FUNCTION_BLOCK OPCUA_WRITE_1322467A4CC663E9C (* Generic Interface Function Block Type *)
  (* Standard: 61499-2 *)
  (* Version 0.0, 01/09/2020, Administrator, nxtControl GmbH, Template *)
  PACKAGE Main;
  (* Compiler Cpp nxtControl builtin 1.0 *)
  {SET_ATTRIBUTE(Runtime.FBType.ImplementingType, Standard.OPCUAClient#DYNGEN_OPCUA_WRITE)}
  {SET_ATTRIBUTE(Configuration.GenericFBType.InterfaceParams, Standard.OPCUAClient#CNTX:=2;VALUE${CNTX$}:BOOL,BOOL)}
  {SET_ATTRIBUTE(Configuration.FBType.IsKind.OPCUA_CLIENT, )}
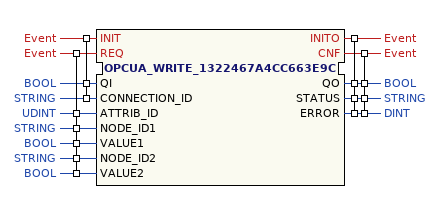
  EVENT_INPUT
    INIT WITH QI, CONNECTION_ID; (* Triggers initialization or deinitialization of FB *)
    REQ WITH ATTRIB_ID, NODE_ID1, NODE_ID2, VALUE1, VALUE2; (* Triggers writing specified node attribute *)
  END_EVENT
  EVENT_OUTPUT
    INITO WITH QO, STATUS, ERROR; (* Confirmation of initialization or deinitialization of FB *)
    CNF WITH QO, STATUS, ERROR; (* Confirmation of completion of write operation *)
  END_EVENT
  VAR_INPUT
    QI : BOOL; (* Qualifier Input. *)
    CONNECTION_ID : STRING; (* Connection  ID associated with server to be accessed *)
    ATTRIB_ID : UDINT; (* Node attribute* ID to be written (13 i.e. node value attribute if not specified) *) {SET_ATTRIBUTE(Configuration.Parameter.DefaultConstant, 13)}
    NODE_ID1 : STRING; (* Node address of node to be accessed (see Node Addressing section for details) *)
    VALUE1 : BOOL; (* Value to be written to specified node attribute *)
    NODE_ID2 : STRING; (* Node address of node to be accessed (see Node Addressing section for details) *)
    VALUE2 : BOOL; (* Value to be written to specified node attribute *)
  END_VAR
  VAR_OUTPUT
    QO : BOOL; (* Output event qualifier *)
    STATUS : STRING; (* Displays status of FB *)
    ERROR : DINT; (* Displays error code for last performed write operation. See section FB Error Codes for description of error codes. *)
  END_VAR
  EC_STATES
    START;
  END_STATES
END_FUNCTION_BLOCK
